// TIA Portal project "001_Integration" (V14)
// Integration of FluidSIM + TIA Portal

(* hardware
DEVICE "S7300/ET200M station_1"  S7-300 station
   slot 0: "Rail_0"  Rail  6ES7 390-1***0-0AA0
   slot 2: "PLC_1"  CPU 314C-2 PN/DP  6ES7 314-6EH04-0AB0  V3.3
      slot 2: "PROFINET interface_1"  PN-IO
         slot 1: "Port_1"  Port
         slot 2: "Port_2"  Port
      slot 5: "DI 24/DO 16_1"  DI24/DO16
      slot 6: "AI 5/AO 2_1"  AI5/AO2
      slot 7: "Count_1"  Counter
      slot 8: "Positioning_1"  Positioning
*)

// ===== PLC "PLC_1"  CPU 314C-2 PN/DP =====

VAR_GLOBAL   // PLC tag table "Memories"
   "Vermelho" AT %M0.1 : Bool;
   "Amarelo" AT %M0.2 : Bool;
   "Verde" AT %M0.3 : Bool;
   "VerdePedestre" AT %M0.4 : Bool;
   "VermelhoPedestre" AT %M0.5 : Bool;
END_VAR

VAR_GLOBAL   // PLC tag table "Lights"
   "StartLight" AT %Q1.0 : Bool;
   "ResetLight" AT %Q1.1 : Bool;
   "AutoLight" AT %Q1.2 : Bool;
   "ManualLight" AT %Q1.3 : Bool;
   "StopLight" AT %Q1.4 : Bool;
END_VAR

VAR_GLOBAL   // PLC tag table "Buttons"
   "StartButton" AT %I1.0 : Bool;
   "StopButton" AT %I1.1 : Bool;
   "Auto_ManSwitch" AT %I1.2 : Bool;
   "ResetButton" AT %I1.3 : Bool;
END_VAR

VAR_GLOBAL   // PLC tag table "Sensors"
   "X1" AT %I0.0 : Bool;
   "X2" AT %I0.1 : Bool;
   "Y1" AT %I0.2 : Bool;
   "Y2" AT %I0.3 : Bool;
   "Y3" AT %I0.4 : Bool;
   "Z1" AT %I0.5 : Bool;
   "Z2" AT %I0.6 : Bool;
END_VAR

VAR_GLOBAL   // PLC tag table "Actuators"
   "X+" AT %Q0.0 : Bool;
   "Y+" AT %Q0.1 : Bool;
   "Y-" AT %Q0.2 : Bool;
   "Z+" AT %Q0.3 : Bool;
   "V" AT %Q0.4 : Bool;
END_VAR

ORGANIZATION_BLOCK "Main"   // OB1, LAD
TITLE = "Main Program Sweep (Cycle)"
{ S7_Optimized_Access := 'FALSE' }
VERSION : 0.1
   VAR_TEMP
      OB1_EV_CLASS : Byte;   // Bits 0-3 = 1 (Coming event), Bits 4-7 = 1 (Event class 1)
      OB1_SCAN_1 : Byte;   // 1 (Cold restart scan 1 of OB 1), 3 (Scan 2-n of OB 1)
      OB1_PRIORITY : Byte;   // Priority of OB Execution
      OB1_OB_NUMBR : Byte;   // 1 (Organization block 1, OB1)
      OB1_RESERVED_1 : Byte;   // Reserved for system
      OB1_RESERVED_2 : Byte;   // Reserved for system
      OB1_PREV_CYCLE : Int;   // Cycle time of previous OB1 scan (milliseconds)
      OB1_MIN_CYCLE : Int;   // Minimum cycle time of OB1 (milliseconds)
      OB1_MAX_CYCLE : Int;   // Maximum cycle time of OB1 (milliseconds)
      OB1_DATE_TIME : Date_And_Time;   // Date and time OB1 started
   END_VAR
BEGIN

REGION Network 1: Enable Machine
   // Ao apertar o botão start, o led de start liga. Ao apertar o Stop ele desliga
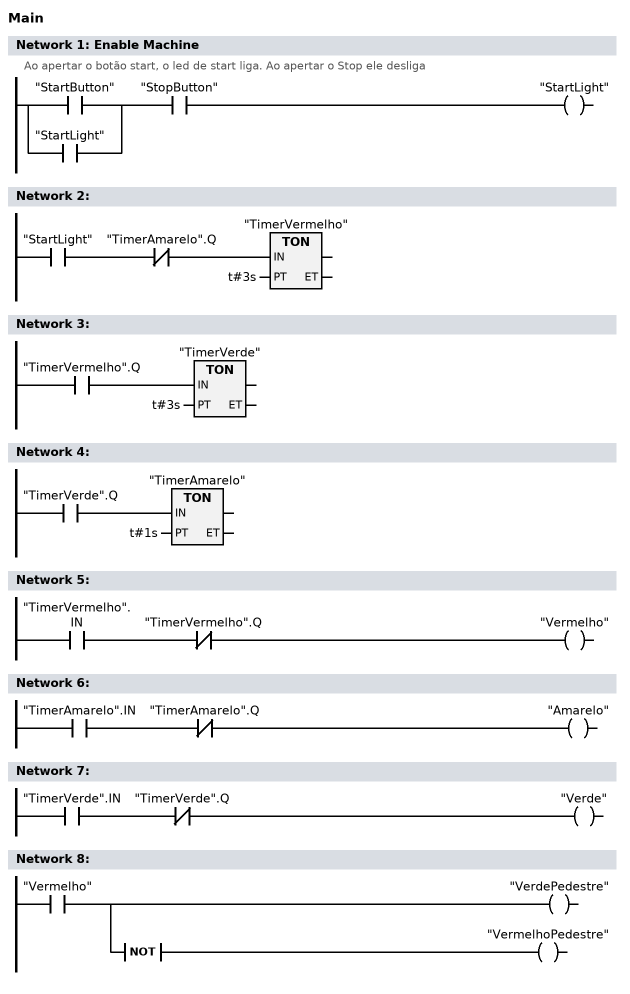
   RUNG wire#powerrail
      Contact( "StartButton" )
      wire#w1
      Contact( "StopButton" )
      Coil( "StartLight" )
   END_RUNG
   RUNG wire#powerrail
      Contact( "StartLight" )
   END_RUNG wire#w1
   // the same network as SCL:
   "StartLight" := ("StartButton" OR "StartLight") AND "StopButton";
END_REGION

REGION Network 2
   "TimerVermelho".TON(IN := "StartLight" AND NOT "TimerAmarelo".Q, PT := t#3s);
END_REGION

REGION Network 3
   "TimerVerde".TON(IN := "TimerVermelho".Q, PT := t#3s);
END_REGION

REGION Network 4
   "TimerAmarelo".TON(IN := "TimerVerde".Q, PT := t#1s);
END_REGION

REGION Network 5
   RUNG wire#powerrail
      Contact( "TimerVermelho".IN )
      I_Contact( "TimerVermelho".Q )
      Coil( "Vermelho" )
   END_RUNG
   // the same network as SCL:
   "Vermelho" := "TimerVermelho".IN AND NOT "TimerVermelho".Q;
END_REGION

REGION Network 6
   RUNG wire#powerrail
      Contact( "TimerAmarelo".IN )
      I_Contact( "TimerAmarelo".Q )
      Coil( "Amarelo" )
   END_RUNG
   // the same network as SCL:
   "Amarelo" := "TimerAmarelo".IN AND NOT "TimerAmarelo".Q;
END_REGION

REGION Network 7
   RUNG wire#powerrail
      Contact( "TimerVerde".IN )
      I_Contact( "TimerVerde".Q )
      Coil( "Verde" )
   END_RUNG
   // the same network as SCL:
   "Verde" := "TimerVerde".IN AND NOT "TimerVerde".Q;
END_REGION

REGION Network 8
   RUNG wire#powerrail
      Contact( "Vermelho" )
      wire#w1
      Coil( "VerdePedestre" )
   END_RUNG
   RUNG wire#w1
      Not()
      Coil( "VermelhoPedestre" )
   END_RUNG
   // the same network as SCL:
   "VerdePedestre" := "Vermelho";
   "VermelhoPedestre" := NOT "Vermelho";
END_REGION
END_ORGANIZATION_BLOCK